// TIA Portal V17 export
// export: Created 2023-04-11T09:34:02.7786761Z, ExportSetting WithDefaults, DisplayName Totally Integrated Automation Portal, DisplayVersion V17 Update 3, DisplayName TIA Portal Openness, DisplayVersion V17 Update 3, DisplayName TIA Portal Version Control Interface, DisplayVersion V17, DisplayName SINAMICS Startdrive Advanced, DisplayVersion V17 Update2, DisplayName SINAMICS Startdrive G130, G150, S120, S150, SINAMICS MV, S210, DisplayVersion V17 Update2, DisplayName SINAMICS Startdrive G110M, G120, G120C, G120D, G120P, G115D, DisplayVersion V17 Update2, DisplayName STEP 7 Professional, DisplayVersion V17 Update 3, DisplayName STEP 7 Safety, DisplayVersion V17, DisplayName WinCC UA Professional, DisplayVersion V17 Update 3
FUNCTION_BLOCK "FB_iTacStdStep"   // FB123, LAD
{ S7_Optimized_Access := 'TRUE' }
VERSION : 0.1
// stored: AutoNumber true, IsIECCheckEnabled false, IsRetainMemResEnabled false, MemoryReserve 100, SetENOAutomatically false, UDAEnableTagReadback false
   VAR_INPUT
      trig : Bool;
      ID : UInt;
      reset : Bool;
      dataDeliminer : String;
      errorText : String;
      errorSignalization : Bool;
      timeout_value : Time;
      DMC : String;
      station : String;
   END_VAR
   VAR_OUTPUT
      pass : Bool;
      fail : Bool;
      exception : Bool;
      timeout_err : Bool;
      retval : UInt;
   END_VAR
   VAR_IN_OUT
      dataToSendIn : "t_LString";
      dataRecieved : "t_LString";
      dataToSendOut : "t_LString";
      rettext_o : String;
   END_VAR
   VAR
      edge : Array[0..0] of Bool;
      Timeout { S7_SetPoint := 'True'} : TON_TIME;
      iPA_iTac_timeout { S7_SetPoint := 'True'} : Program_Alarm;
      iPA_iTac_fail { S7_SetPoint := 'True'} : Program_Alarm;
      toutErr : Bool;
      retValStr : String;
      dataReady : Bool;
      ID_1 { ExternalAccessible := 'False'; ExternalVisible := 'False'; ExternalWritable := 'False'} : "t_LString";
   END_VAR
   VAR_TEMP
      id_x : UInt;
      id_x1 : Bool;
      id_x9 : Bool;
      fail_local : Bool;
      pass_local : Bool;
      auxStr : String;
      ID_recieved : UInt;
      sendPLS : Bool;
   END_VAR
   VAR_TEMP   // added for the SCL form of the ladder/FBD networks
      _w1 : Bool;
      _w2 : Bool;
      _w3 : Bool;
   END_VAR
BEGIN

REGION Network 1: reset / init
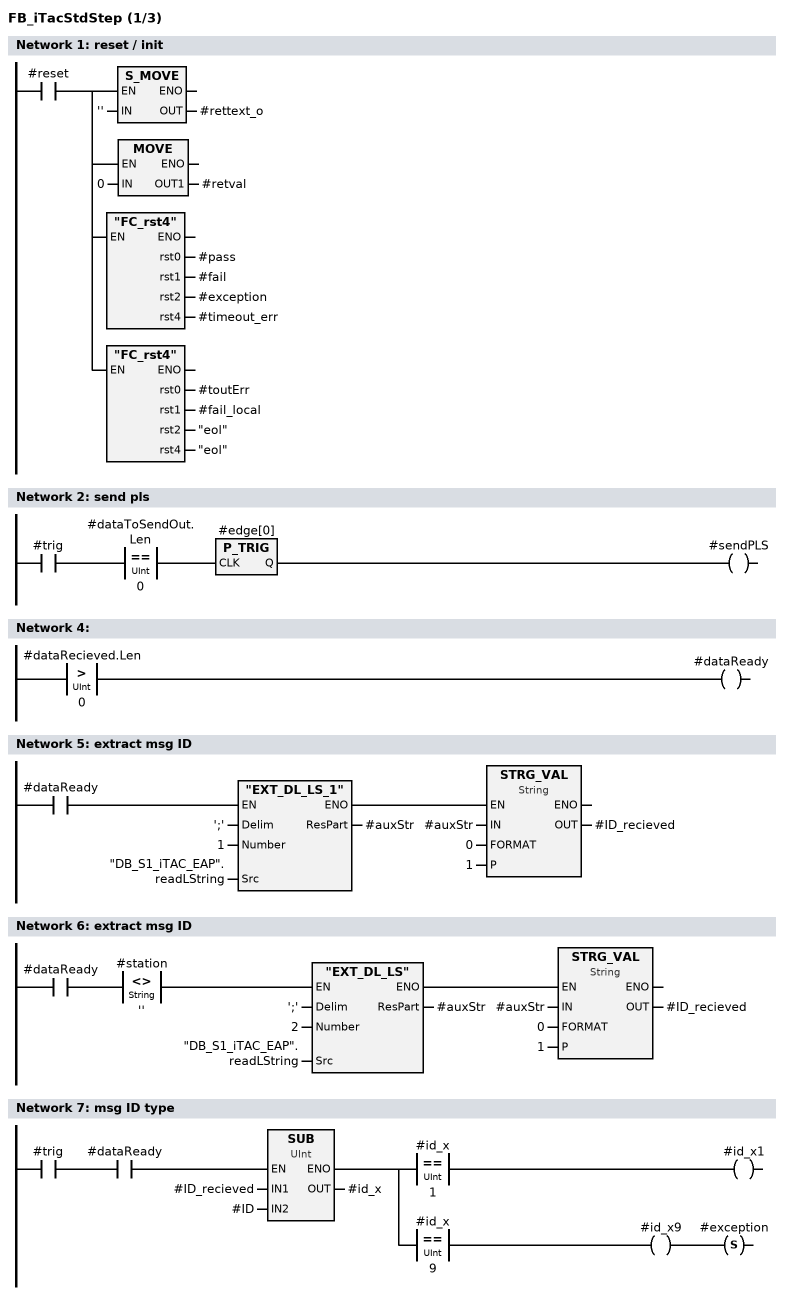
   RUNG wire#powerrail
      Contact( #reset )
      wire#w1
      S_Move(in := '', out => #rettext_o)
   END_RUNG
   RUNG wire#w1
      Move(in := 0, out1 => #retval)
   END_RUNG
   RUNG wire#w1
      "FC_rst4"(rst0 => #pass, rst1 => #fail, rst2 => #exception, rst4 => #timeout_err)
   END_RUNG
   RUNG wire#w1
      "FC_rst4"(rst0 => #toutErr, rst1 => #fail_local, rst2 => "eol", rst4 => "eol")
   END_RUNG
   // the same network as SCL:
   IF #reset THEN
       #rettext_o := '';
       #retval := 0;
       "FC_rst4"(rst0 => #pass, rst1 => #fail, rst2 => #exception, rst4 => #timeout_err);
       "FC_rst4"(rst0 => #toutErr, rst1 => #fail_local, rst2 => "eol", rst4 => "eol");
   END_IF;
END_REGION

REGION Network 2: send pls
   RUNG wire#powerrail
      Contact( #trig )
      { S7_Templates := "SrcType := UInt" } EQ_Contact(in1 := #dataToSendOut.Len, in2 := 0)
      P_Trig( #edge[0] )
      Coil( #sendPLS )
   END_RUNG
   // the same network as SCL:
   #_w1 := #trig AND (#dataToSendOut.Len = 0);
   #_w2 := #_w1 AND NOT #edge[0];   // rising edge
   #edge[0] := #_w1;
   #sendPLS := #_w2;
END_REGION

REGION Network 3 (SCL): prepare send data
   IF #sendPLS THEN

       // add station
       "TO_LS_1"(IN := #station,
                 OUT := #dataToSendOut);
       // copy ID
       "CONCAT_LS_1"(IN1 := #dataToSendOut,
                     IN2 := #dataDeliminer,
                     OUT := #dataToSendOut);

       "TO_LS_1"(IN := #ID, OUT := #ID_1);
       "CONCAT_LS_LS_1"(IN1 := #dataToSendOut,
                        IN2 := #ID_1,
                        OUT := #dataToSendOut);
       // add DMC data
       IF (#DMC <> '') THEN

           "CONCAT_LS_1"(IN1 := #dataToSendOut,
                       IN2 := #dataDeliminer,
                       OUT := #dataToSendOut);

           "CONCAT_LS_1"(IN1 := #dataToSendOut,
                         IN2 := #DMC,
                         OUT := #dataToSendOut);
       END_IF;

       // add other data
       IF (#dataToSendIn.Len<> 0) THEN

           "CONCAT_LS_1"(IN1 := #dataToSendOut,
                       IN2 := #dataDeliminer,
                       OUT := #dataToSendOut);

           "CONCAT_LS_LS_1"(IN1 := #dataToSendOut,
                          IN2 := #dataToSendIn,
                       OUT := #dataToSendOut);
       END_IF;

   END_IF;
END_REGION

REGION Network 4
   RUNG wire#powerrail
      { S7_Templates := "SrcType := UInt" } GT_Contact(in1 := #dataRecieved.Len, in2 := 0)
      Coil( #dataReady )
   END_RUNG
   // the same network as SCL:
   #dataReady := #dataRecieved.Len > 0;
END_REGION

REGION Network 5: extract msg ID
   RUNG wire#powerrail
      Contact( #dataReady )
      "EXT_DL_LS_1"(Delim := ';', Number := 1, Src := "DB_S1_iTAC_EAP".readLString, ResPart => #auxStr)
      { S7_Templates := "[src_type := String, dest_type := UInt]" } STRG_VAL(IN := #auxStr, FORMAT := 0, P := 1, OUT => #ID_recieved)
   END_RUNG
   // the same network as SCL:
   "EXT_DL_LS_1"(EN := #dataReady,
                 Delim := ';',
                 Number := 1,
                 Src := "DB_S1_iTAC_EAP".readLString,
                 ResPart => #auxStr,
                 ENO => #_w1);
   IF #_w1 THEN STRG_VAL(IN := #auxStr, FORMAT := 0, P := 1, OUT => #ID_recieved); END_IF;
END_REGION

REGION Network 6: extract msg ID
   RUNG wire#powerrail
      Contact( #dataReady )
      { S7_Templates := "SrcType := String" } NE_Contact(in1 := #station, in2 := '')
      "EXT_DL_LS"(Delim := ';', Number := 2, Src := "DB_S1_iTAC_EAP".readLString, ResPart => #auxStr)
      { S7_Templates := "[src_type := String, dest_type := UInt]" } STRG_VAL(IN := #auxStr, FORMAT := 0, P := 1, OUT => #ID_recieved)
   END_RUNG
   // the same network as SCL:
   "EXT_DL_LS"(EN := #dataReady AND (#station <> ''),
               Delim := ';',
               Number := 2,
               Src := "DB_S1_iTAC_EAP".readLString,
               ResPart => #auxStr,
               ENO => #_w1);
   IF #_w1 THEN STRG_VAL(IN := #auxStr, FORMAT := 0, P := 1, OUT => #ID_recieved); END_IF;
END_REGION

REGION Network 7: msg ID type
   RUNG wire#powerrail
      Contact( #trig )
      Contact( #dataReady )
      { S7_Templates := "SrcType := UInt" } Sub(in1 := #ID_recieved, in2 := #ID, out => #id_x)
      wire#w1
      { S7_Templates := "SrcType := UInt" } EQ_Contact(in1 := #id_x, in2 := 1)
      Coil( #id_x1 )
   END_RUNG
   RUNG wire#w1
      { S7_Templates := "SrcType := UInt" } EQ_Contact(in1 := #id_x, in2 := 9)
      Coil( #id_x9 )
      S_Coil( #exception )
   END_RUNG
   // the same network as SCL:
   #_w1 := #trig AND #dataReady;
   IF #_w1 THEN #id_x := #ID_recieved - #ID; END_IF;
   #id_x1 := #_w1 AND (#id_x = 1);
   #id_x9 := #_w1 AND (#id_x = 9);
   IF #id_x9 THEN #exception := TRUE; END_IF;
END_REGION

REGION Network 8: pass or fail
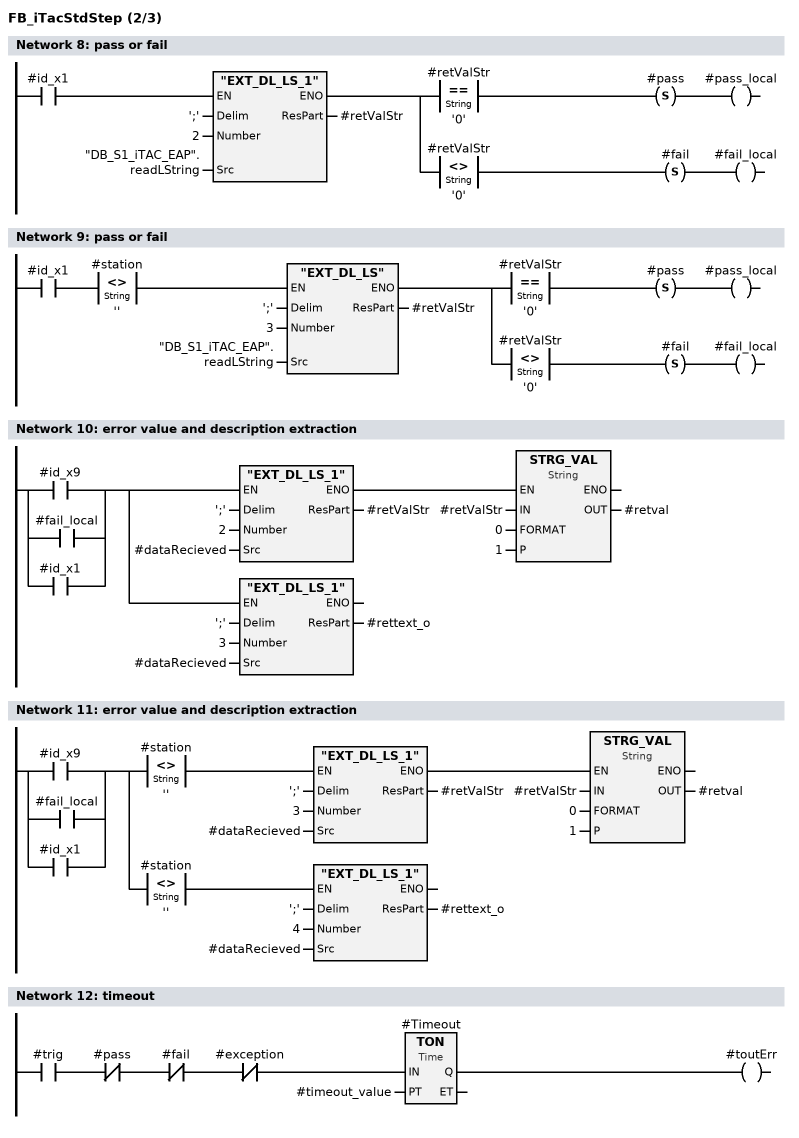
   RUNG wire#powerrail
      Contact( #id_x1 )
      "EXT_DL_LS_1"(Delim := ';', Number := 2, Src := "DB_S1_iTAC_EAP".readLString, ResPart => #retValStr)
      wire#w1
      { S7_Templates := "SrcType := String" } EQ_Contact(in1 := #retValStr, in2 := '0')
      S_Coil( #pass )
      Coil( #pass_local )
   END_RUNG
   RUNG wire#w1
      { S7_Templates := "SrcType := String" } NE_Contact(in1 := #retValStr, in2 := '0')
      S_Coil( #fail )
      Coil( #fail_local )
   END_RUNG
   // the same network as SCL:
   "EXT_DL_LS_1"(EN := #id_x1,
                 Delim := ';',
                 Number := 2,
                 Src := "DB_S1_iTAC_EAP".readLString,
                 ResPart => #retValStr,
                 ENO => #_w1);
   #_w2 := #_w1 AND (#retValStr = '0');
   IF #_w2 THEN #pass := TRUE; END_IF;
   #pass_local := #_w2;
   #_w3 := #_w1 AND (#retValStr <> '0');
   IF #_w3 THEN #fail := TRUE; END_IF;
   #fail_local := #_w3;
END_REGION

REGION Network 9: pass or fail
   RUNG wire#powerrail
      Contact( #id_x1 )
      { S7_Templates := "SrcType := String" } NE_Contact(in1 := #station, in2 := '')
      "EXT_DL_LS"(Delim := ';', Number := 3, Src := "DB_S1_iTAC_EAP".readLString, ResPart => #retValStr)
      wire#w1
      { S7_Templates := "SrcType := String" } EQ_Contact(in1 := #retValStr, in2 := '0')
      S_Coil( #pass )
      Coil( #pass_local )
   END_RUNG
   RUNG wire#w1
      { S7_Templates := "SrcType := String" } NE_Contact(in1 := #retValStr, in2 := '0')
      S_Coil( #fail )
      Coil( #fail_local )
   END_RUNG
   // the same network as SCL:
   "EXT_DL_LS"(EN := #id_x1 AND (#station <> ''),
               Delim := ';',
               Number := 3,
               Src := "DB_S1_iTAC_EAP".readLString,
               ResPart => #retValStr,
               ENO => #_w1);
   #_w2 := #_w1 AND (#retValStr = '0');
   IF #_w2 THEN #pass := TRUE; END_IF;
   #pass_local := #_w2;
   #_w3 := #_w1 AND (#retValStr <> '0');
   IF #_w3 THEN #fail := TRUE; END_IF;
   #fail_local := #_w3;
END_REGION

REGION Network 10: error value and description extraction
   RUNG wire#powerrail
      Contact( #id_x9 )
      wire#w1
      "EXT_DL_LS_1"(Delim := ';', Number := 2, Src := #dataRecieved, ResPart => #retValStr)
      { S7_Templates := "[src_type := String, dest_type := UInt]" } STRG_VAL(IN := #retValStr, FORMAT := 0, P := 1, OUT => #retval)
   END_RUNG
   RUNG wire#powerrail
      Contact( #fail_local )
   END_RUNG wire#w1
   RUNG wire#powerrail
      Contact( #id_x1 )
   END_RUNG wire#w1
   RUNG wire#w1
      "EXT_DL_LS_1"(Delim := ';', Number := 3, Src := #dataRecieved, ResPart => #rettext_o)
   END_RUNG
   // the same network as SCL:
   "EXT_DL_LS_1"(EN := #id_x9 OR #fail_local OR #id_x1,
                 Delim := ';',
                 Number := 2,
                 Src := #dataRecieved,
                 ResPart => #retValStr,
                 ENO => #_w1);
   IF #_w1 THEN STRG_VAL(IN := #retValStr, FORMAT := 0, P := 1, OUT => #retval); END_IF;
   IF #id_x9 OR #fail_local OR #id_x1 THEN
       "EXT_DL_LS_1"(Delim := ';', Number := 3, Src := #dataRecieved, ResPart => #rettext_o);
   END_IF;
END_REGION

REGION Network 11: error value and description extraction
   RUNG wire#powerrail
      Contact( #id_x9 )
      wire#w1
      { S7_Templates := "SrcType := String" } NE_Contact(in1 := #station, in2 := '')
      "EXT_DL_LS_1"(Delim := ';', Number := 3, Src := #dataRecieved, ResPart => #retValStr)
      { S7_Templates := "[src_type := String, dest_type := UInt]" } STRG_VAL(IN := #retValStr, FORMAT := 0, P := 1, OUT => #retval)
   END_RUNG
   RUNG wire#powerrail
      Contact( #fail_local )
   END_RUNG wire#w1
   RUNG wire#powerrail
      Contact( #id_x1 )
   END_RUNG wire#w1
   RUNG wire#w1
      { S7_Templates := "SrcType := String" } NE_Contact(in1 := #station, in2 := '')
      "EXT_DL_LS_1"(Delim := ';', Number := 4, Src := #dataRecieved, ResPart => #rettext_o)
   END_RUNG
   // the same network as SCL:
   #_w1 := #id_x9 OR #fail_local OR #id_x1;
   "EXT_DL_LS_1"(EN := #_w1 AND (#station <> ''),
                 Delim := ';',
                 Number := 3,
                 Src := #dataRecieved,
                 ResPart => #retValStr,
                 ENO => #_w2);
   IF #_w2 THEN STRG_VAL(IN := #retValStr, FORMAT := 0, P := 1, OUT => #retval); END_IF;
   IF #_w1 AND (#station <> '') THEN
       "EXT_DL_LS_1"(Delim := ';', Number := 4, Src := #dataRecieved, ResPart => #rettext_o);
   END_IF;
END_REGION

REGION Network 12: timeout
   RUNG wire#powerrail
      Contact( #trig )
      I_Contact( #pass )
      I_Contact( #fail )
      I_Contact( #exception )
      { S7_Templates := "time_type := Time" } #Timeout.TON(pt := #timeout_value, et =>)
      Coil( #toutErr )
   END_RUNG
   // the same network as SCL:
   #Timeout(IN := #trig AND NOT #pass AND NOT #fail AND NOT #exception, PT := #timeout_value);   // TON
   #toutErr := #Timeout.Q;
END_REGION

REGION Network 13: raise timeout error
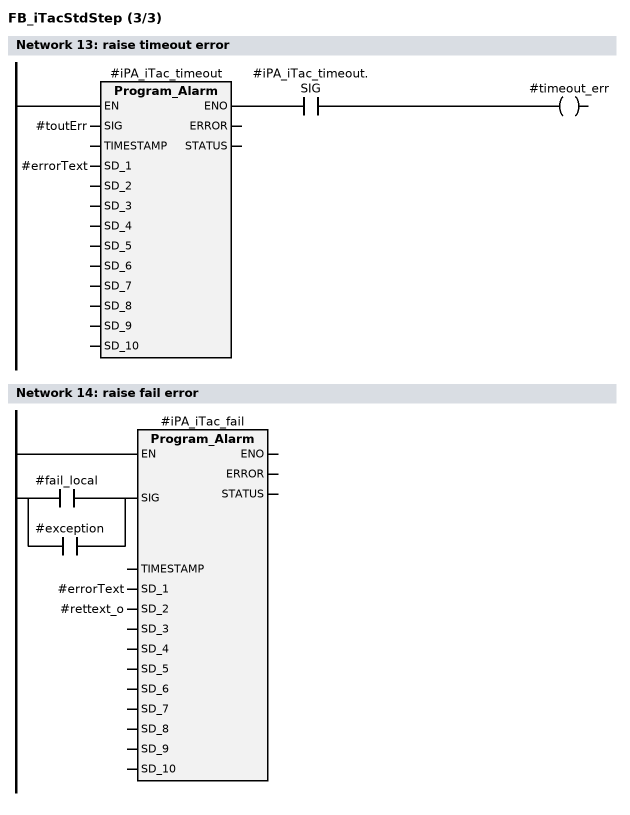
   RUNG wire#powerrail
      #iPA_iTac_timeout.Program_Alarm(SIG := #toutErr, TIMESTAMP :=, SD_1 := #errorText, SD_2 :=, SD_3 :=, SD_4 :=, SD_5 :=, SD_6 :=, SD_7 :=, SD_8 :=, SD_9 :=, SD_10 :=, Error =>, Status =>)
      Contact( #iPA_iTac_timeout.SIG )
      Coil( #timeout_err )
   END_RUNG
   // the same network as SCL:
   #iPA_iTac_timeout(SIG := #toutErr, SD_1 := #errorText, ENO => #_w1);   // Program_Alarm
   #timeout_err := #_w1 AND #iPA_iTac_timeout.SIG;
END_REGION

REGION Network 14: raise fail error
   RUNG wire#powerrail
      #iPA_iTac_fail.Program_Alarm(SIG := wire#w1, TIMESTAMP :=, SD_1 := #errorText, SD_2 := #rettext_o, SD_3 :=, SD_4 :=, SD_5 :=, SD_6 :=, SD_7 :=, SD_8 :=, SD_9 :=, SD_10 :=, Error =>, Status =>)
   END_RUNG
   RUNG wire#powerrail
      Contact( #fail_local )
   END_RUNG wire#w1
   RUNG wire#powerrail
      Contact( #exception )
   END_RUNG wire#w1
   // the same network as SCL:
   #iPA_iTac_fail(SIG := #fail_local OR #exception, SD_1 := #errorText, SD_2 := #rettext_o);   // Program_Alarm
END_REGION
END_FUNCTION_BLOCK
